(* PLC project Unnamed, Unknown Unnamed 1 *)
(* stored: creationDateTime 2023-06-26T21:38:42, modificationDateTime 2023-07-06T02:37:00 *)

PROGRAM program0
  VAR
    AtScaleEntry AT %IX100.0 : BOOL;
    AtScale AT %IX100.1 : BOOL;
    AtScaleExit AT %IX100.2 : BOOL;
    AtLeftEntry AT %IX100.3 : BOOL;
    AtExitLeft AT %IX100.4 : BOOL;
    AtForwardEntry AT %IX100.5 : BOOL;
    AtRightEntry AT %IX100.7 : BOOL;
    Start AT %IX101.1 : BOOL;
    Reset AT %IX101.2 : BOOL;
    Stop AT %IX101.3 : BOOL;
    EmergencyStop AT %IX101.4 : BOOL;
    EntryConveyor AT %QX100.0 : BOOL;
    LoadScale AT %QX100.1 : BOOL;
    SendLeft AT %QX100.2 : BOOL;
    LeftConveyor AT %QX100.3 : BOOL;
    SendRight AT %QX100.4 : BOOL;
    RightConveyor AT %QX100.5 : BOOL;
    SendForward AT %QX100.6 : BOOL;
    FrontConveyor AT %QX100.7 : BOOL;
    StartLight AT %QX101.0 : BOOL;
    ResetLight AT %QX101.1 : BOOL;
    StopLight AT %QX101.2 : BOOL;
    Weight AT %IW100 : INT;
    LeftCount AT %QW100 : INT;
    ForwardCount AT %QW101 : INT;
    RightCount AT %QW102 : INT;
    WeightCounter AT %QW103 : INT;
  END_VAR
  VAR
    TP0 : TP;
    TON0 : TON;
    TON1 : TON;
    TON2 : TON;
    CTU0 : CTU;
    CTU1 : CTU;
    CTU2 : CTU;
  END_VAR
  VAR  (* added by the conversion: wires and edge detectors of the diagram *)
    _GT116_ENO : BOOL;
    _GT116_OUT : BOOL;
    _LE119_ENO : BOOL;
    _LE119_OUT : BOOL;
    _GT16_ENO : BOOL;
    _GT16_OUT : BOOL;
    _LE20_ENO : BOOL;
    _LE20_OUT : BOOL;
    _GE123_ENO : BOOL;
    _GE123_OUT : BOOL;
    R_TRIG1 : R_TRIG;
    R_TRIG2 : R_TRIG;
    R_TRIG3 : R_TRIG;
  END_VAR

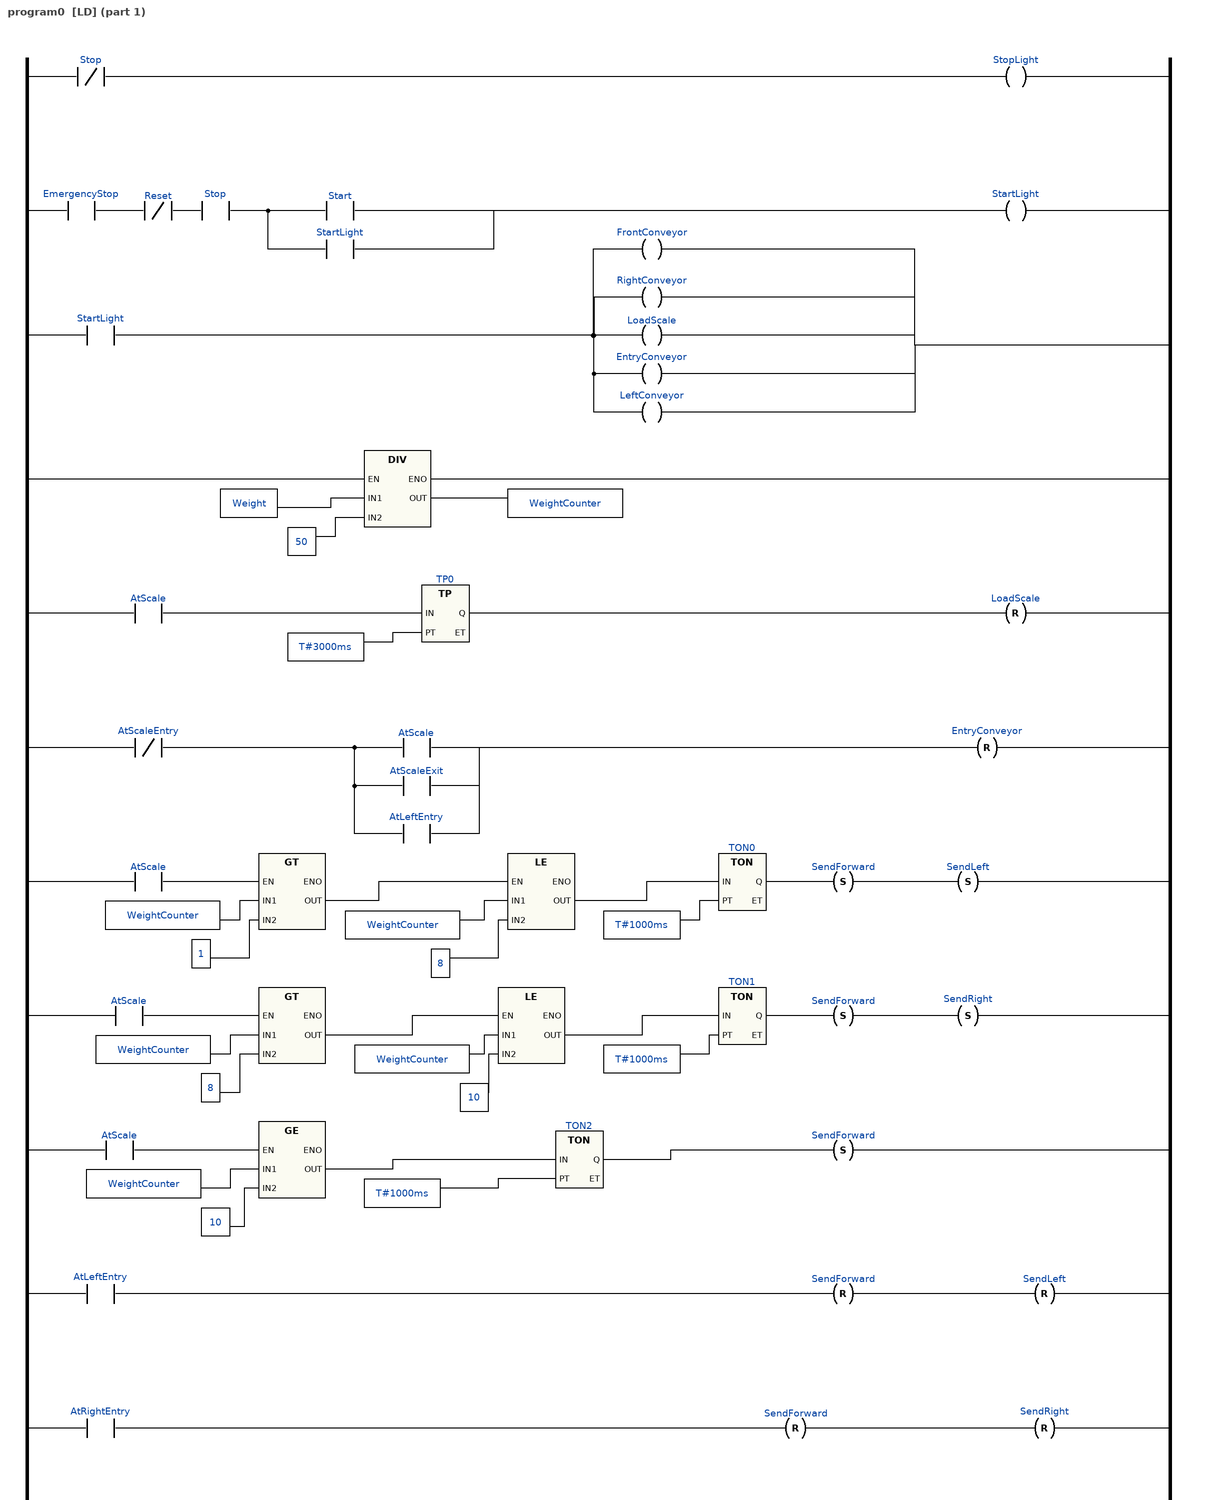
(* LD diagram, written out as Structured Text *)
StopLight := NOT Stop;
StartLight := EmergencyStop AND NOT Reset AND Stop AND (Start OR StartLight);
FrontConveyor := StartLight;
RightConveyor := StartLight;
LoadScale := StartLight;
EntryConveyor := StartLight;
LeftConveyor := StartLight;
WeightCounter := Weight / 50;
TP0(IN := AtScale, PT := T#3000ms);
IF TP0.Q THEN LoadScale := FALSE; END_IF;
IF NOT AtScaleEntry AND (AtScale OR AtScaleExit OR AtLeftEntry) THEN EntryConveyor := FALSE; END_IF;
_GT116_OUT := GT(EN := AtScale, IN1 := WeightCounter, IN2 := 1, ENO => _GT116_ENO);
_LE119_OUT := LE(EN := _GT116_OUT, IN1 := WeightCounter, IN2 := 8, ENO => _LE119_ENO);
TON0(IN := _LE119_OUT, PT := T#1000ms);
IF TON0.Q THEN SendForward := TRUE; END_IF;
IF TON0.Q THEN SendLeft := TRUE; END_IF;
_GT16_OUT := GT(EN := AtScale, IN1 := WeightCounter, IN2 := 8, ENO => _GT16_ENO);
_LE20_OUT := LE(EN := _GT16_OUT, IN1 := WeightCounter, IN2 := 10, ENO => _LE20_ENO);
TON1(IN := _LE20_OUT, PT := T#1000ms);
IF TON1.Q THEN SendForward := TRUE; END_IF;
IF TON1.Q THEN SendRight := TRUE; END_IF;
_GE123_OUT := GE(EN := AtScale, IN1 := WeightCounter, IN2 := 10, ENO => _GE123_ENO);
TON2(IN := _GE123_OUT, PT := T#1000ms);
IF TON2.Q THEN SendForward := TRUE; END_IF;
IF AtLeftEntry THEN SendForward := FALSE; END_IF;
IF AtLeftEntry THEN SendLeft := FALSE; END_IF;
IF AtRightEntry THEN SendForward := FALSE; END_IF;
IF AtRightEntry THEN SendRight := FALSE; END_IF;
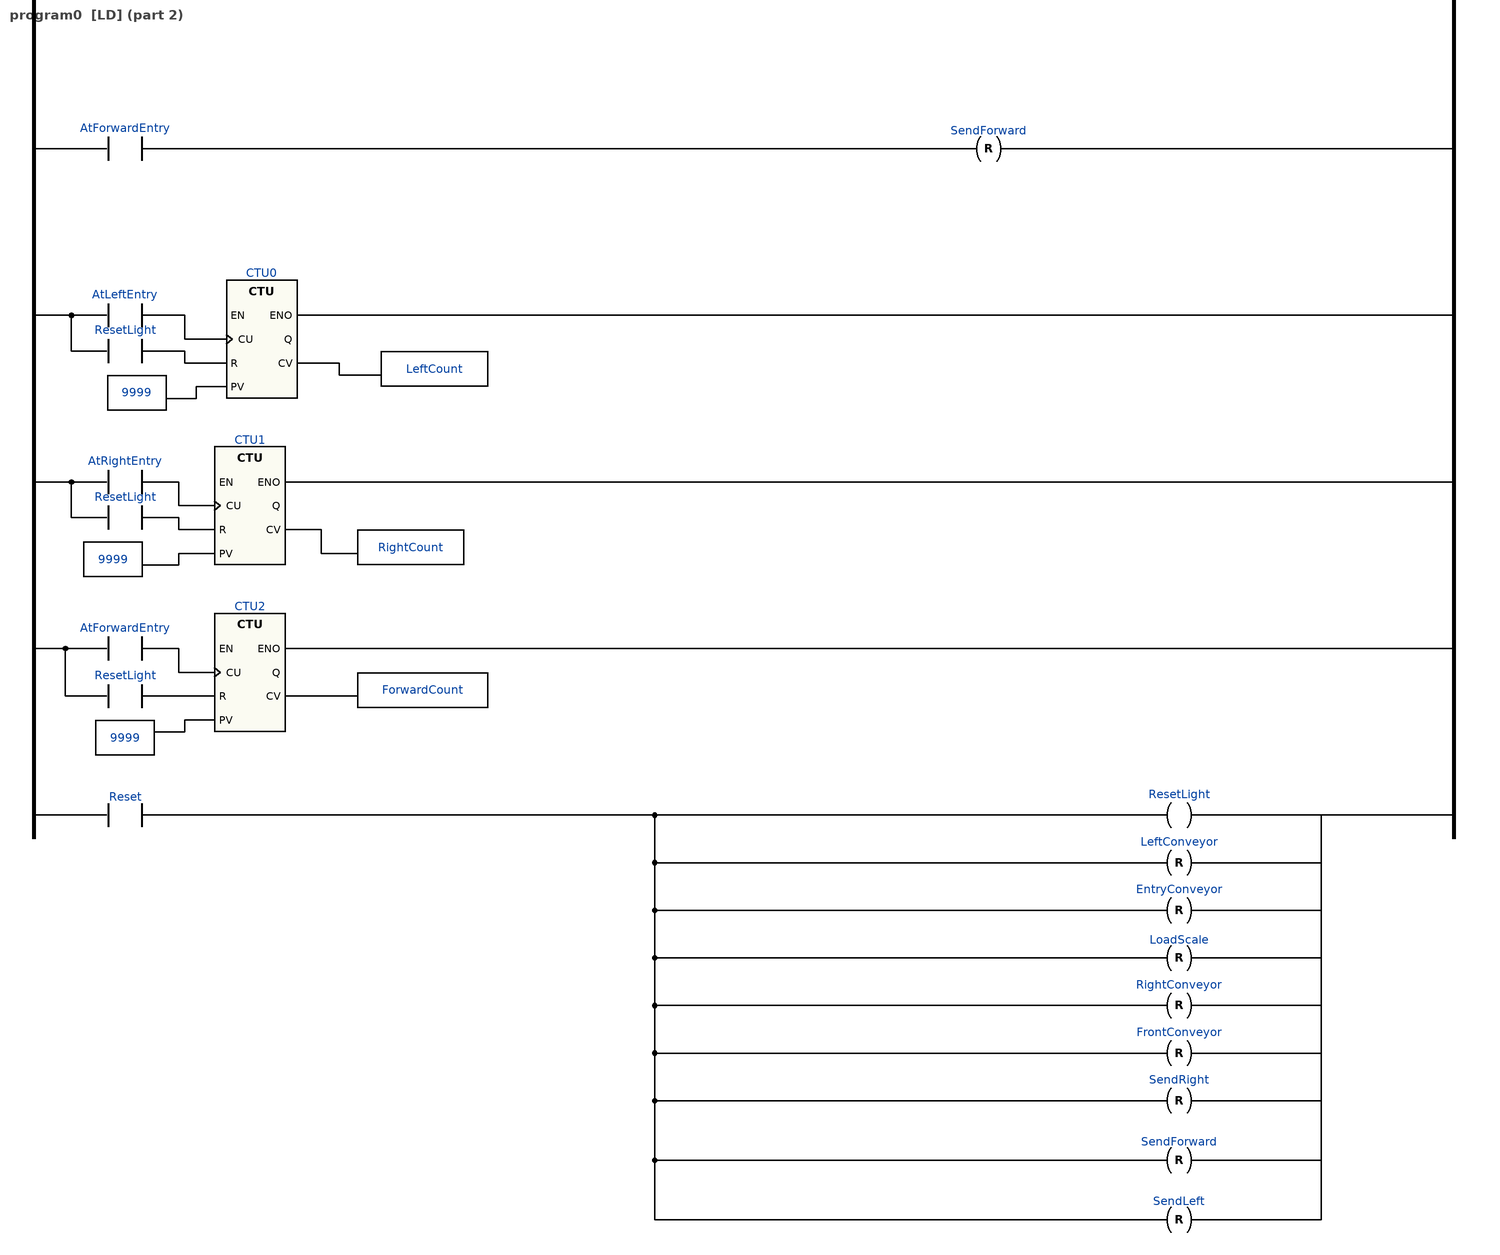
IF AtForwardEntry THEN SendForward := FALSE; END_IF;
R_TRIG1(CLK := AtLeftEntry);
CTU0(CU := R_TRIG1.Q, R := ResetLight, PV := 9999);
LeftCount := CTU0.CV;
R_TRIG2(CLK := AtRightEntry);
CTU1(CU := R_TRIG2.Q, R := ResetLight, PV := 9999);
RightCount := CTU1.CV;
R_TRIG3(CLK := AtForwardEntry);
CTU2(CU := R_TRIG3.Q, R := ResetLight, PV := 9999);
ForwardCount := CTU2.CV;
ResetLight := Reset;
IF Reset THEN LeftConveyor := FALSE; END_IF;
IF Reset THEN EntryConveyor := FALSE; END_IF;
IF Reset THEN LoadScale := FALSE; END_IF;
IF Reset THEN RightConveyor := FALSE; END_IF;
IF Reset THEN FrontConveyor := FALSE; END_IF;
IF Reset THEN SendRight := FALSE; END_IF;
IF Reset THEN SendForward := FALSE; END_IF;
IF Reset THEN SendLeft := FALSE; END_IF;
END_PROGRAM

CONFIGURATION Config0
  RESOURCE Res0 ON PLC
    TASK task0(INTERVAL := T#20ms, PRIORITY := 0);
    PROGRAM instance0 WITH task0 : program0;
  END_RESOURCE
END_CONFIGURATION
